INTERFACE I_ExternControl_Process

METHOD PUBLIC DelBitDWord : DWORD
VAR_INPUT
  inVal   : DWORD;
  bitNo   : DWORD;
END_VAR
END_METHOD

PROPERTY EnableProcess : dword
GET
END_GET
SET
END_SET
END_PROPERTY

METHOD PUBLIC GetBitDWord : BOOL
VAR_INPUT
  inVal   : DWORD;
  bitNo   : DINT;
END_VAR
END_METHOD

METHOD PUBLIC Init : BOOL
END_METHOD

PROPERTY MoverCountInQueue : uint
GET
END_GET
END_PROPERTY

PROPERTY MoverInQueue : Bool
GET
END_GET
END_PROPERTY

PROPERTY ProcessCmd : E_STATION_CTRL
SET
END_SET
END_PROPERTY

PROPERTY ProcessPerMinute : uint
GET
END_GET
END_PROPERTY

PROPERTY ProcessState : E_STATION_STATE
GET
END_GET
END_PROPERTY

PROPERTY ProcessType : e_process_type
GET
END_GET
SET
END_SET
END_PROPERTY

METHOD PUBLIC SetBitDWord : DWORD
VAR_INPUT
  inVal   : DWORD;
  bitNo   : DWORD;
END_VAR
END_METHOD

METHOD PUBLIC SetBitWord : WORD
VAR_INPUT
  inVal   : WORD;
  bitNo   : DINT;
END_VAR
END_METHOD

PROPERTY StationCount : uint
GET
END_GET
END_PROPERTY

PROPERTY StationFirst : uint
GET
END_GET
SET
END_SET
END_PROPERTY

PROPERTY TargetMask : dword
GET
END_GET
SET
END_SET
END_PROPERTY

END_INTERFACE

(* stored: Version 1.1.0.1, ProductVersion 3.1.4024.12
   Itf I_ExternControl_Process: Id {1e0151f7-eebc-4938-aa9d-dfc7c8d50a0e}
   Folder properties: Id {d0801dd2-1fe3-4f74-8a18-68fad6ff0850}
   Folder public: Id {885a99d6-b473-49ea-ab53-4e7138e0c618}
   Method DelBitDWord: Id {5cb7e06f-3da9-4a1a-bea5-9a988ffc7f17}
   Property EnableProcess: Id {9699bf5e-2077-4cb7-99fc-c0847193d1a9}
   Get Get: Id {0c619069-ad6d-44f1-b2dd-39896ec58416}
   Set Set: Id {1841a1fb-e3a6-4734-9435-52faead727cc}
   Method GetBitDWord: Id {df2afb96-c7e2-4b2d-a08a-0c1377859704}
   Method Init: Id {8e726022-9386-41d3-92bc-e79944b82059}
   Property MoverCountInQueue: Id {fb14633e-f6ba-42fc-b863-34843086f547}
   Get Get: Id {fd64fcfc-3520-47a0-ae34-fbdc9d3b9dd7}
   Property MoverInQueue: Id {9c7c6232-d39a-43f3-9d58-49cbcf18c9e6}
   Get Get: Id {4b69c1a8-dbe8-4273-b733-8b21afdbfc6d}
   Property ProcessCmd: Id {878ce26f-61d4-44ae-9d2f-6c47be4c28ef}
   Set Set: Id {f9f726b6-05c3-4294-8279-b0c68ebe8b61}
   Property ProcessPerMinute: Id {3c6b74ac-8016-4f8e-b93b-4a6adf586768}
   Get Get: Id {826d8484-ddbe-48fe-aa84-07f643c39bcb}
   Property ProcessState: Id {6b18f165-f4a0-4383-afee-672cf6b7e001}
   Get Get: Id {f5049e5f-416c-4194-bb2b-222124e685de}
   Property ProcessType: Id {37a018c4-d4db-4578-acc2-c447c8063402}
   Get Get: Id {7e54a6da-33b9-457c-997c-18e7d30cc287}
   Set Set: Id {7b12e57b-907b-4366-b6c7-7585cc658d8e}
   Method SetBitDWord: Id {0af7c71c-a6b4-49bb-a415-8a6aed0768f9}
   Method SetBitWord: Id {8633b640-5090-458e-a471-4b35825b9c02}
   Property StationCount: Id {c090c780-c0ea-4ba7-88fb-1d66b20d11df}
   Get Get: Id {8ba734cb-4c5c-4eb3-a5e0-96141c1387aa}
   Property StationFirst: Id {7fed964a-d10e-418c-b30e-864e4bf5564a}
   Get Get: Id {49451648-355d-4fe9-9fed-605def6d2c8c}
   Set Set: Id {a7412949-fc97-42d5-8be1-e6a3fb1b293b}
   Property TargetMask: Id {220bef15-bc98-48b2-a7fe-cd5cc154f97e}
   Get Get: Id {bc8900b8-e5df-4d0f-adf9-300c795befaa}
   Set Set: Id {31e29fe5-f8b6-4115-9df9-c421e88efe82} *)
